(* IEC 61131-3 sources: template-app/template/test, 1 file *)

(* ---- dummy.st ---- *)
USING AxUnit.Assert;
{TestFixture}
CLASS MyTestFixture
    VAR PRIVATE
        x : BOOL := TRUE;
    END_VAR
    {Test}
    METHOD PUBLIC MyTestMethod
        Equal(actual := x, expected := TRUE);
    END_METHOD
END_CLASS
